FUNCTION WRITE_PROTECTED_LREAL : BOOL
VAR_INPUT
    ptr: POINTER TO LREAL;
    val: LREAL;
END_VAR

ptr^ := val;

END_FUNCTION

(* stored: Version 1.1.0.1, ProductVersion 3.1.4022.9
   POU WRITE_PROTECTED_LREAL: Id {339c1152-50eb-418b-b2b4-54330f145c79}, SpecialFunc None *)
